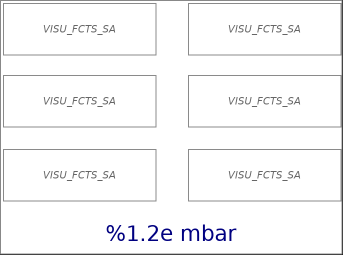
VISUALIZATION SA_POMP_1E_PCR_PPM  // 343x255
VAR_IN_OUT
	m_Input_PRG:		BLOCK_PRG_POMPAGE;
	m_Input_Jauge:		BLOCK_BCG450_ANA;
END_VAR
    Rectangle (0,0 343x255)
    Frame (3,75 153x52)
        shows VISU_FCTS_SA(m_Input_ID_XML := 0, m_Input_UserRight := PRG_USER.ACTU_USER.FONCTION_SA, m_Input_Operation := m_Input_PRG.POMPAGE.OP_Pompage_Sec)
    Frame (3,3 153x52)
        shows VISU_FCTS_SA(m_Input_ID_XML := 1, m_Input_UserRight := PRG_USER.ACTU_USER.FONCTION_SA, m_Input_Operation := m_Input_PRG.POMPAGE.OP_Marche_Pompes)
    Frame (188,3 153x52)
        shows VISU_FCTS_SA(m_Input_ID_XML := 2, m_Input_UserRight := PRG_USER.ACTU_USER.FONCTION_SA, m_Input_Operation := m_Input_PRG.POMPAGE.OP_Arret_Pompes)
    Frame (188,75 153x52)
        shows VISU_FCTS_SA(m_Input_ID_XML := 3, m_Input_UserRight := PRG_USER.ACTU_USER.FONCTION_SA, m_Input_Operation := m_Input_PRG.POMPAGE.OP_Isolement)
    Frame (3,149 153x52)
        shows VISU_FCTS_SA(m_Input_ID_XML := 4, m_Input_UserRight := PRG_USER.ACTU_USER.FONCTION_SA, m_Input_Operation := m_Input_PRG.POMPAGE.OP_Ventilation)
    Rectangle (80,219 182x29), "%1.2e mbar", text variable: m_Input_Jauge.STATE_Pression
    Frame (188,149 153x52)
        shows VISU_FCTS_SA(m_Input_ID_XML := 17, m_Input_UserRight := PRG_USER.ACTU_USER.FONCTION_SA, m_Input_Operation := m_Input_PRG.POMPAGE.OP_Regen)
END_VISUALIZATION

(* stored: Version 1.1.0.1, ProductVersion 3.1.4024.10
   Visu SA_POMP_1E_PCR_PPM: Id {f7f44d04-cee1-483f-b5ec-f3d6f60c58f6} *)
